Yaskawa INFORM job: hand_blower_cylinder_program.JBI

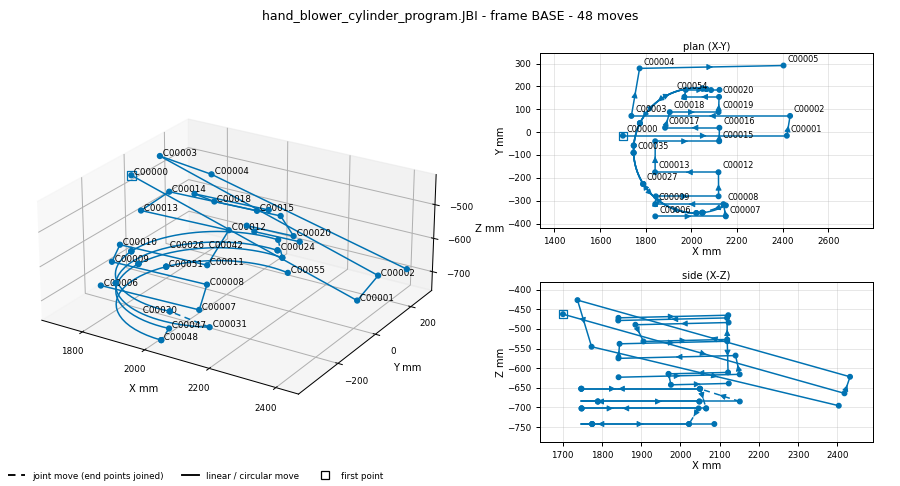
[picture p0: tool path of hand_blower_cylinder_program.JBI in frame BASE, 48 of 63 moves have a stored position in this frame; points joined in program order, loops and branches not executed]
/JOB
//NAME hand_blower_cylinder_program
//POS
///NPOS 56,0,56,0,0,0
///TOOL 0
///POSTYPE BASE
///RECTAN
///RCONF 0,0,0,0,0,0,0,0,0,0,0,0,0,0,0,0,0,0,0,0,0,0,0,0
C00000=1700.589821,-15.984108,-462.500019,175.000000,-44.616549,106.561944
C00001=2417.740168,-15.984108,-664.206933,175.000000,-44.616549,106.561944
C00002=2431.967717,70.671298,-622.031680,-167.105484,14.987914,5.000000
C00003=1737.629674,70.671298,-426.740992,-167.105484,14.987914,5.000000
C00004=1773.507288,278.674345,-545.479908,175.000000,-66.363125,-97.070806
C00005=2403.308036,291.162907,-695.721300,175.000000,-60.000000,-97.070806
C00006=1842.258005,-368.684770,-623.185813,175.000000,-60.000000,89.599473
C00007=2150.765321,-368.684925,-615.823660,175.000000,-60.000000,89.599473
C00008=2140.319490,-315.438119,-567.978259,175.000000,-52.280236,88.942392
C00009=1841.935020,-315.437969,-575.098842,175.000000,-52.280236,88.942392
C00010=1844.758913,-281.084604,-538.063237,175.000000,-41.933679,88.477719
C00011=2119.163093,-281.084741,-531.514914,175.000000,-41.933679,88.477719
C00012=2118.656282,-175.573916,-472.036278,-163.089074,-5.000000,-5.000000
C00013=1841.418330,-175.573778,-478.652225,-163.089074,-5.000000,-5.000000
C00014=1841.901234,-40.186135,-471.837803,168.843166,-5.000000,5.000000
C00015=2121.795946,-40.186276,-465.158456,168.843166,-5.000000,5.000000
C00016=2122.608103,18.950861,-483.808995,156.106630,-5.000000,5.000000
C00017=1885.165789,18.950980,-489.475268,156.106630,-5.000000,5.000000
C00018=1905.619017,87.288208,-532.004906,175.000000,-40.502295,-88.399054
C00019=2119.093847,87.288101,-526.910588,175.000000,-40.502295,-88.399054
C00020=2121.215661,154.028853,-610.926129,175.000000,-62.616769,-89.291780
C00021=1969.591171,154.028929,-614.544464,175.000000,-62.616769,-89.291780
C00022=1975.689802,184.626965,-642.504701,175.000000,-60.000000,-89.851834
C00023=2123.085266,184.626891,-638.987287,175.000000,-60.000000,-89.851834
C00024=2048.166540,190.553939,-685.006500,84.133594,-90.000000,5.000000
C00025=2048.166540,190.553939,-685.006500,84.133594,-90.000000,5.000000
C00026=1776.536610,42.078019,-685.006500,153.189413,-90.000000,5.000000
C00027=1789.477237,-227.071618,-685.006500,-147.684128,-89.999999,5.000000
C00028=1789.477237,-227.071618,-685.006500,-147.684128,-89.999999,5.000000
C00029=1789.477237,-227.071618,-685.006500,-147.684128,-89.999999,5.000000
C00030=1949.621259,-344.870476,-685.006500,-104.990839,-90.000000,5.000000
C00031=2151.141007,-320.753216,-685.006500,-61.360114,-90.000000,5.000000
C00032=2049.328751,-352.611910,-652.508460,-175.000000,-60.000000,96.111597
C00033=2049.328751,-352.611910,-652.508460,-175.000000,-60.000000,96.111597
C00034=1861.847521,-303.522445,-652.508460,175.000000,-60.000000,54.542916
C00035=1747.352332,-90.738104,-652.508460,175.000000,-60.000000,5.000000
C00036=1747.352332,-90.738104,-652.508460,175.000000,-60.000000,5.000000
C00037=1747.352332,-90.738104,-652.508460,175.000000,-60.000000,5.000000
C00038=1834.348104,118.929361,-652.508460,175.000000,-60.000000,-47.094110
C00039=2050.112371,190.346962,-652.508460,175.000000,-60.000000,-96.276980
C00040=2065.368795,188.231848,-702.560960,175.000000,-60.000000,-99.509094
C00041=2065.368795,188.231848,-702.560960,175.000000,-60.000000,-99.509094
C00042=1847.828505,130.660434,-702.560960,175.000000,-60.000000,-50.844237
C00043=1748.097135,-58.750506,-702.560960,175.000000,-60.000000,-5.000000
C00044=1748.097135,-58.750506,-702.560960,175.000000,-60.000000,-5.000000
C00045=1748.097135,-58.750506,-702.560960,175.000000,-60.000000,-5.000000
C00046=1851.533754,-295.804337,-702.560960,175.000000,-60.000000,51.839817
C00047=2046.135968,-352.934810,-702.560960,175.000000,-60.000000,95.438274
C00048=2021.692934,-354.160168,-742.361460,-175.000000,-60.000000,90.301530
C00049=2021.692934,-354.160168,-742.361460,-175.000000,-60.000000,90.301530
C00050=1759.871741,-163.367117,-742.361460,175.000000,-60.000000,17.535695
C00051=1774.887437,38.758948,-742.361460,175.000000,-60.000000,-26.032952
C00052=1774.887437,38.758948,-742.361460,175.000000,-60.000000,-26.032952
C00053=1774.887437,38.758948,-742.361460,175.000000,-60.000000,-26.032952
C00054=1919.666435,172.782424,-742.361460,-175.000000,-60.000000,-68.385521
C00055=2086.267529,183.885268,-742.361460,175.000000,-60.000000,-103.988996
///POSTYPE PULSE
///PULSE
EX00000=181248.0
EX00001=275456.0
EX00002=306176.0
///POSTYPE PULSE
///PULSE
EC00000=181248.0
EC00001=181248.0
EC00002=181248.0
EC00003=181248.0
EC00004=181248.0
EC00005=181248.0
EC00006=275456.0
EC00007=275456.0
EC00008=275456.0
EC00009=275456.0
EC00010=275456.0
EC00011=275456.0
EC00012=275456.0
EC00013=275456.0
EC00014=275456.0
EC00015=275456.0
EC00016=275456.0
EC00017=275456.0
EC00018=275456.0
EC00019=275456.0
EC00020=275456.0
EC00021=275456.0
EC00022=275456.0
EC00023=275456.0
EC00024=306176.0
EC00025=306176.0
EC00026=306176.0
EC00027=306176.0
EC00028=306176.0
EC00029=306176.0
EC00030=306176.0
EC00031=306176.0
EC00032=306176.0
EC00033=306176.0
EC00034=306176.0
EC00035=306176.0
EC00036=306176.0
EC00037=306176.0
EC00038=306176.0
EC00039=306176.0
EC00040=306176.0
EC00041=306176.0
EC00042=306176.0
EC00043=306176.0
EC00044=306176.0
EC00045=306176.0
EC00046=306176.0
EC00047=306176.0
EC00048=306176.0
EC00049=306176.0
EC00050=306176.0
EC00051=306176.0
EC00052=306176.0
EC00053=306176.0
EC00054=306176.0
EC00055=306176.0
//INST
///DATE 2023/08/16 17:04
///ATTR SC,RW,RJ
////FRAME BASE
///GROUP1 RB1,ST1
NOP
MOVJ P009 EX000 VJ=15.00
MOVJ C00000 EC00000 VJ=15.0
CALL JOB:SPYON
MOVL C00001 EC00001 V=150.0
MOVL C00002 EC00002 V=150.0
MOVL C00003 EC00003 V=150.0
MOVL C00004 EC00004 V=150.0
MOVL C00005 EC00005 V=150.0
CALL JOB:SPYOF
MOVJ P009 VJ=15.00
MOVL P009 EX00000 V=150.0
MOVJ C00006 EC00006 VJ=15.0
CALL JOB:SPYON
MOVL C00007 EC00007 V=150.0
MOVL C00008 EC00008 V=150.0
MOVL C00009 EC00009 V=150.0
MOVL C00010 EC00010 V=150.0
MOVL C00011 EC00011 V=150.0
MOVL C00012 EC00012 V=150.0
MOVL C00013 EC00013 V=150.0
MOVL C00014 EC00014 V=150.0
MOVL C00015 EC00015 V=150.0
MOVL C00016 EC00016 V=150.0
MOVL C00017 EC00017 V=150.0
MOVL C00018 EC00018 V=150.0
MOVL C00019 EC00019 V=150.0
MOVL C00020 EC00020 V=150.0
MOVL C00021 EC00021 V=150.0
MOVL C00022 EC00022 V=150.0
MOVL C00023 EC00023 V=150.0
CALL JOB:SPYOF
MOVJ P009 VJ=15.00
MOVL P009 EX00001 V=150.0
MOVJ C00024 EC00024 VJ=15.0
CALL JOB:SPYON
MOVC C00025 EC00025 V=150.0
MOVC C00026 EC00026 V=150.0
MOVC C00027 EC00027 V=150.0
MOVJ C00028 EC00028 VJ=15.0
MOVC C00029 EC00029 V=150.0
MOVC C00030 EC00030 V=150.0
MOVC C00031 EC00031 V=150.0
MOVJ C00032 EC00032 VJ=15.0
MOVC C00033 EC00033 V=150.0
MOVC C00034 EC00034 V=150.0
MOVC C00035 EC00035 V=150.0
MOVJ C00036 EC00036 VJ=15.0
MOVC C00037 EC00037 V=150.0
MOVC C00038 EC00038 V=150.0
MOVC C00039 EC00039 V=150.0
MOVJ C00040 EC00040 VJ=15.0
MOVC C00041 EC00041 V=150.0
MOVC C00042 EC00042 V=150.0
MOVC C00043 EC00043 V=150.0
MOVJ C00044 EC00044 VJ=15.0
MOVC C00045 EC00045 V=150.0
MOVC C00046 EC00046 V=150.0
MOVC C00047 EC00047 V=150.0
MOVJ C00048 EC00048 VJ=15.0
MOVC C00049 EC00049 V=150.0
MOVC C00050 EC00050 V=150.0
MOVC C00051 EC00051 V=150.0
MOVJ C00052 EC00052 VJ=15.0
MOVC C00053 EC00053 V=150.0
MOVC C00054 EC00054 V=150.0
MOVC C00055 EC00055 V=150.0
CALL JOB:SPYOF
MOVJ P009 VJ=15.00
MOVL P009 EX00002 V=150.0
END
